ABB RAPID module: TCP_MF.MOD

MODULE TCP_MF
	! Points are read in order of declaration.
  ! Please do not change the order of points!

  LOCAL PERS robtarget pTCP_Point1:=[[466.2944,-290.5074,295.5301],[0.313281178474426,0.278983324766159,0.90399032831192,-0.082611508667469],[-1,0,0,0],[9E+09,9E+09,9E+09,9E+09,9E+09,9E+09]];
	LOCAL PERS robtarget pTCP_Point2:=[[447.7713,-354.7118,284.1492],[0.230896160006523,0.555310547351837,0.796820163726807,0.058264221996069],[-1,0,0,0],[9E+09,9E+09,9E+09,9E+09,9E+09,9E+09]];
	LOCAL PERS robtarget pTCP_Point3:=[[490.5464,-274.994,293.5444],[0.216596066951752,-0.178762018680573,0.958910286426544,-0.0402662083506584],[-1,0,-1,0],[9E+09,9E+09,9E+09,9E+09,9E+09,9E+09]];
	LOCAL PERS robtarget pTCP_Point4:=[[446.4561,-190.6827,240.9932],[0.0964178666472435,-0.578861355781555,0.769202947616577,-0.252883166074753],[-1,0,-2,1],[9E+09,9E+09,9E+09,9E+09,9E+09,9E+09]];

ENDMODULE
